// TIA Portal V17 export
// export: Created 2025-03-10T12:17:50.652005Z, ExportSetting WithDefaults, DisplayName Totally Integrated Automation Portal, DisplayVersion V17 Update 8, DisplayName TIA Portal Openness, DisplayVersion V17 Update 8, DisplayName TIA Portal Version Control Interface, DisplayVersion V17, DisplayName SINAMICS Startdrive Advanced, DisplayVersion V17 SP2, DisplayName SINAMICS Startdrive G110M, G120, G120C, G120D, G120P, G115D, DisplayVersion V17 SP2, DisplayName SINAMICS Startdrive G130, G150, S120, S150, SINAMICS MV, S210, DisplayVersion V17 SP2, DisplayName STEP 7 Professional, DisplayVersion V17 Update 8, DisplayName SINUMERIK ONE STEP 7 Toolbox, DisplayVersion V17 Update 12, DisplayName SINUMERIK 840D sl STEP 7 Toolbox, DisplayVersion V17 Update 12, DisplayName STEP 7 Safety, DisplayVersion V17 Update 6, DisplayName WinCC Advanced, DisplayVersion V17 Update 8
TYPE "AXIS"
// stored: IsFailsafeCompliant false
   STRUCT
      ENABLED : Bool;   // ENABLED
      SELECTED : Bool;   // SELECTED
      HMI_JOG_MINUS_RQ : Bool;   // HMI JOG MINUS RQ
      HMI_JOG_PLUS_RQ : Bool;   // HMI JOG PLUS RQ
      HMI_JOG_MINUS_CMM : Bool;   // HMI JOG MINUS COMMAND
      HMI_JOG_PLUS_CMM : Bool;   // HMI JOG PLUS COMMAND
      AUTO_RETURN_CMM : Bool;   // AUTO RETURN COMMAND
      AUTO_ADVANCE_CMM : Bool;   // AUTO ADVANCE COMMAND
      JOG_HELP : Bool;   // JOG HELP
      MINUS_BUTTON_HELP : Bool;   // MINUS BUTTON HELP
      PLUS_BUTTON_HELP : Bool;   // PLUS BUTTON HELP
      OPERATOR_HELP : Bool;   // OPERATOR HELP
      P1_TRIGGER : Bool;   // P1 TRIGGER
      P2_TRIGGER : Bool;   // P2 TRIGGER
      N1_TRIGGER : Bool;   // N1 TRIGGER
      N2_TRIGGER : Bool;   // N2 TRIGGER
      POS_TO_GO_FC18 : Real;   // POS TO GO FC18
      FC18_AXIS_IN_POS : Bool;   // FC18 AXIS IN POSITION
      FC18_FAULT : Bool;   // FC18 FAULT
      E_GANT_GROUP_SYN : Bool;   // GANTRY GROUP IS SYNCRONOUS
   END_STRUCT;
END_TYPE
